Universal Robots PolyScope program: TEST_ROTSUP.urp

Program TEST_ROTSUP (installation=GD directory=/programs/GD createdIn=5.13.0 lastSavedIn=5.13.0 robotSerialNumber=20205000017)
Calibrated DH parameters: a=[-0.000157, -0.56303, -0.236706, -0.000074, -0.000109, 0]; d=[0.181705, 47.632387, 369.599619, -417.058513, 0.119878, 0.115667]; alpha=[1.570881, -0.005074, -0.001247, 1.56886, -1.570997, 0]; deltaTheta=[0, -0.405485, 5.544791, 1.143886, -0.000009, -0.000001]
InitVariablesNode
BeforeStart
  Script file /programs/GD/CONTROL/FORCE_CONTROL.script
    | def GET_TCP_FORCE_TOOL():
    |   force_torque=get_tcp_force()
    |   force_B=p[force_torque[0], force_torque[1], force_torque[2], 0, 0, 0]
    |   torque_B=p[force_torque[3], force_torque[4], force_torque[5], 0, 0, 0]
    |   tcp=get_actual_tcp_pose()
    |   rotation_BT=p[0, 0, 0, tcp[3], tcp[4], tcp[5]]
    |   force_T=pose_trans(pose_inv(rotation_BT), force_B)
    |   torque_T=pose_trans(pose_inv(rotation_BT), torque_B)
    |   force_torque_T=p[force_T[0], force_T[1], force_T[2], torque_T[0], torque_T[1], torque_T[2]]
    |   return force_torque_T
    | end
    | 
    | def GET_FORCE_VALUE_RZ(target):
    |   PoseSub= pose_sub (CurrPos_p,target)
    |   RZSub=r2d(PoseSub[5])
    |   if (PoseSub[5]>=0):
    |     RZMin=RZSupDegMin
    |     RZForceVal=RZSupForceVal
    |   else:
    |     RZMin=-RZSupDegMin
    |     RZForceVal=-RZSupForceVal
    |   end
    |   if (r2d(norm(PoseSub[5])) >= RZSupDegMin):
    |     return (RZMin-RZSub)*RZSupForceRatio+RZForceVal
    |   else:
    |     return 0
    |   end
    | end
Robot Program (runOnlyOnce=true)
  SetPayload (workpieceName=k2)
  Wait Sleep waitTime=0.02
  SuppressedNode
    Force Frame feature=Joint_6_name; selection=[1, 1, 1, 1, 1, 1]; wrench=[0, 0, 0, 0, 0, -1]; limitsForce=[0.01, 0.01, 0.015, 0.174533, 0.174533, 0.087266]; limitsMotion=[0.1, 0.1, 0.1, 0.349066, 0.349066, 0.349066]
      Wait Sleep waitTime=10
  SuppressedNode
    Popup Message (haltProgram=false message=111 inputType=Text)
  Script: zero_ftsensor()
  ForceStep := 1
  SuppressedNode
    ForceFeature := p[0,0,0,0,0,0]
  ForceFeature := tool_pose()
  var_1 := 0
  SuppressedNode
    var_2 := [0,0,1,0,0,1]
  var_2 := [1,1,1,1,1,1]
  var_3 := 2
  Script: ForceValue[2]=-20
  Script: ForceValue[5]=1
  ForceLimit := [0.01,0.01,ForceLimitZ[ForceStep-1],d2r(10.),d2r(10.),d2r(10.)]
  Script: force_mode(ForceFeature,var_2,ForceValue,var_3,ForceLimit)
  Loop Counting (count=100000) loopVariable(name=ループ_1)
    If UseRZSuppress
      SuppressedNode
        If WorkPosNo≟0 removedSiblings(If(type=ElseIf checkContinuously=false, expression=WorkPosNo≟1, children(Script(type=Line, expression=ForceValue[5]=GET_FORCE_VALUE_RZ(g1GD_pos5)))))
          Script: ForceValue[5]=GET_FORCE_VALUE_RZ(g2GD_pos5)
      SuppressedNode
        Script: ForceValue[5]=GET_FORCE_VALUE_RZ(TEST_ROTSUP)
      Script: var_1=GET_FORCE_VALUE_RZ(TEST_ROTSUP)
      var_4 := ForceValue
      Script: var_4[5]=var_1
      SuppressedNode
        If norm(RZSub)>15
          Script: break
      Script: force_mode(ForceFeature,var_2,var_4,var_3,ForceLimit)
      SuppressedNode
        Script: force_mode(ForceFeature,var_2,ForceValue,var_3,ForceLimit)
    Script: sync()
  Script: end_force_mode()
  Script: stopl(5.0)
  Popup Message (haltProgram=false message=! inputType=Text)
  SetPayload (workpieceName=k10)
Thread スレッド_1 (runOnlyOnce=false)
  Script: CurrPos=get_actual_tool_flange_pose()
  Script: CurrPos_p=get_actual_tcp_pose()
  Script: sync()
